ABB RobotStudio station: Project2.rsstnx

Station Project2 (saved by RobotStudio 24.3.10885.0)
Controller Controller1
  mechanical unit ROB_1: IRB2600_12_185__02, 6 joints, base frame (0, 0, 0) mm
Layout (positions relative to the parent item):
  - Ratata [mechanism] at (1018.61, 0, 1417.5) mm, rotated rx 180 ry 60 rz 180 deg
      TCP Ratata at (0, -50, 190) mm, rotated rx 30 ry 0 rz 0 deg
      links: Group_2
  - IRB2600_12_185__02 [mechanism, from %ABB.RobotStudio.Models.IRB2600%\IRB2600_12_185_G_02.rslib] at (0, 0, 0) mm; joint values [0, 0, 0, 0, 0.5236, 0] (rad or m)
  - Part_6 [part], size 214.9 x 213.7 x 0 mm
  - Part_7 [part] at (135.15, 0, 0) mm, size 214.9 x 213.7 x 400 mm
  - Part_14 [part], size 168 x 171.3 x 400 mm
  - Part_16 [part] at (400, 920.93, 1412.57) mm, rotated rx 0 ry 90 rz 0 deg, size 214.9 x 213.7 x 400 mm
  - Part_17 [part], size 1500 x 10 x 1500 mm
Attachment: Ratata is attached to IRB2600_12_185__02 / Link6
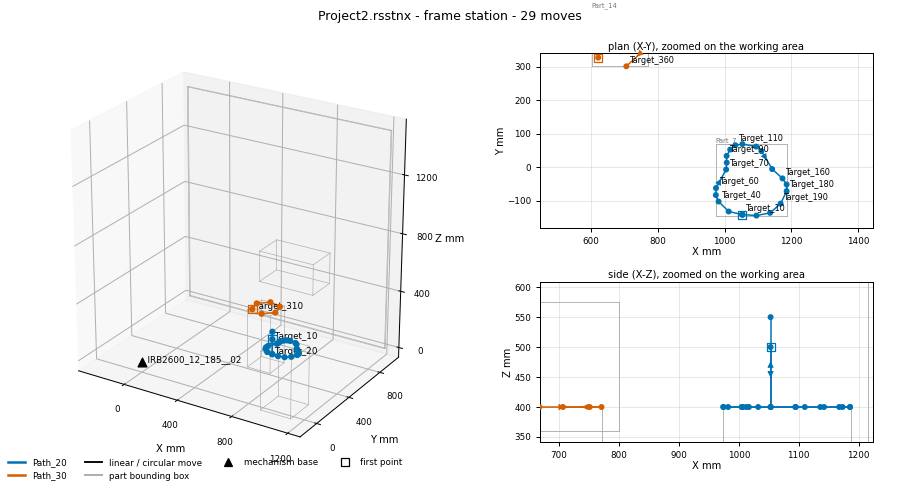
[picture p0: tool path of Project2.rsstnx in frame station, 29 of 29 moves have a stored position in this frame; points joined in program order, loops and branches not executed]
Targets, tools, work objects and paths stored in the station, written as RAPID:
! task T_ROB1
MODULE CalibData
  PERS tooldata Ratata:=[TRUE,[[0,-50,190],[0.965925826,0.258819045,0,0]],[1,[0,0,90],[1,0,0,0],0,0,0]];
  TASK PERS wobjdata Workobject_1:=[FALSE,TRUE,"",[[622.473,327.081,400],[1,0,0,0]],[[0,0,0],[1,0,0,0]]];
ENDMODULE

! task T_ROB1
MODULE Module1
  CONST jointtarget JointTarget_1:=[[0,0,0,0,0,0],[9E+09,9E+09,9E+09,9E+09,9E+09,9E+09]];
  CONST robtarget Target_10:=[[1053.028483888,-141.83,500],[0,0.048639314,0.998816408,0],[0,0,0,0],[9E+09,9E+09,9E+09,9E+09,9E+09,9E+09]];
  CONST robtarget Target_20:=[[1053.028483888,-141.83,400],[0,0.048639314,0.998816408,0],[-1,0,-1,0],[9E+09,9E+09,9E+09,9E+09,9E+09,9E+09]];
  CONST robtarget Target_30:=[[1012.393593189,-132.667043204,400],[0,0.247498073,0.968888386,0],[-1,0,-1,0],[9E+09,9E+09,9E+09,9E+09,9E+09,9E+09]];
  CONST robtarget Target_40:=[[982.192356429,-102.911473019,400],[0,0.483619111,0.875278559,0],[-1,0,-1,0],[9E+09,9E+09,9E+09,9E+09,9E+09,9E+09]];
  CONST robtarget Target_50:=[[973.974019148,-83.529915198,400],[0,0.630396667,0.776273175,0],[-1,1,-1,0],[9E+09,9E+09,9E+09,9E+09,9E+09,9E+09]];
  CONST robtarget Target_60:=[[974.486081612,-62.744242155,400],[0,0.783865496,0.620930659,0],[-1,2,-2,0],[9E+09,9E+09,9E+09,9E+09,9E+09,9E+09]];
  CONST robtarget Target_70:=[[1004.654113735,-7.369996452,400],[0,0.83364436,0.552301621,0],[0,3,-2,0],[9E+09,9E+09,9E+09,9E+09,9E+09,9E+09]];
  CONST robtarget Target_80:=[[1006.554953292,13.24883335,400],[0,0.617780056,0.786350941,0],[-1,1,-1,0],[9E+09,9E+09,9E+09,9E+09,9E+09,9E+09]];
  CONST robtarget Target_90:=[[1006.144920769,33.417655307,400],[0,0.829177231,0.558985796,0],[0,3,-2,0],[9E+09,9E+09,9E+09,9E+09,9E+09,9E+09]];
  CONST robtarget Target_100:=[[1016.902942171,52.408008378,400],[0,0.878010395,0.478641563,0],[0,3,-2,0],[9E+09,9E+09,9E+09,9E+09,9E+09,9E+09]];
  CONST robtarget Target_110:=[[1032.336239923,65.35895098,400],[0,0.986205127,0.165527784,0],[0,3,-2,0],[9E+09,9E+09,9E+09,9E+09,9E+09,9E+09]];
  CONST robtarget Target_120:=[[1053.446161766,68.778243604,400],[0,0.99965304,0.026340074,0],[0,3,-2,0],[9E+09,9E+09,9E+09,9E+09,9E+09,9E+09]];
  CONST robtarget Target_130:=[[1094.310928385,61.39343752,400],[0,0.971088832,-0.238718412,0],[0,3,-2,0],[9E+09,9E+09,9E+09,9E+09,9E+09,9E+09]];
  CONST robtarget Target_140:=[[1110.161148991,47.833471517,400],[0,0.897820327,-0.440361966,0],[0,3,-2,0],[9E+09,9E+09,9E+09,9E+09,9E+09,9E+09]];
  CONST robtarget Target_150:=[[1142.282150365,-5.867956748,400],[0,0.940674196,-0.33931115,0],[0,3,-2,0],[9E+09,9E+09,9E+09,9E+09,9E+09,9E+09]];
  CONST robtarget Target_160:=[[1173.132567714,-33.754311671,400],[0,0.896740471,-0.442556808,0],[0,3,-2,0],[9E+09,9E+09,9E+09,9E+09,9E+09,9E+09]];
  CONST robtarget Target_170:=[[1185.623777539,-51.793265608,400],[0,0.845978482,-0.533217036,0],[-1,3,-2,0],[9E+09,9E+09,9E+09,9E+09,9E+09,9E+09]];
  CONST robtarget Target_180:=[[1185.639297263,-71.745848185,400],[0,-0.586154613,0.810199216,0],[-1,4,-1,0],[9E+09,9E+09,9E+09,9E+09,9E+09,9E+09]];
  CONST robtarget Target_190:=[[1167.562709351,-109.141891193,400],[0,-0.422507005,0.906359658,0],[-1,4,-1,0],[9E+09,9E+09,9E+09,9E+09,9E+09,9E+09]];
  CONST robtarget Target_200:=[[1136.030927079,-136.731454767,400],[0,-0.222736348,0.97487872,0],[-1,4,-1,0],[9E+09,9E+09,9E+09,9E+09,9E+09,9E+09]];
  CONST robtarget Target_210:=[[1095.203821678,-144.904989424,400],[0,-0.003413263,0.999994175,0],[-1,4,-1,0],[9E+09,9E+09,9E+09,9E+09,9E+09,9E+09]];
  CONST robtarget Target_220:=[[1053.028483888,-141.83,400],[0,0.048639314,0.998816408,0],[0,0,0,0],[9E+09,9E+09,9E+09,9E+09,9E+09,9E+09]];
  CONST robtarget Target_230:=[[1053.028483888,-141.83,550],[0,0.048639314,0.998816408,0],[0,0,0,0],[9E+09,9E+09,9E+09,9E+09,9E+09,9E+09]];
  CONST robtarget Target_290:=[[-19.683,85.658,0],[0,1,0,0],[0,0,0,0],[9E+09,9E+09,9E+09,9E+09,9E+09,9E+09]];
  CONST robtarget Target_300:=[[560.683986041,-377.081,922.5],[0.482962913,0.129409523,0.836516304,-0.224143868],[0,-1,0,0],[9E+09,9E+09,9E+09,9E+09,9E+09,9E+09]];
  CONST robtarget Target_310:=[[0,0,0],[0,0.622915127,0.782289425,0],[0,0,0,0],[9E+09,9E+09,9E+09,9E+09,9E+09,9E+09]];
  CONST robtarget Target_320:=[[-19.683271052,85.657574479,0],[0,0.622915127,0.782289425,0],[0,0,0,0],[9E+09,9E+09,9E+09,9E+09,9E+09,9E+09]];
  CONST robtarget Target_330:=[[44.656728948,145.532574479,0],[0,0.930605037,0.366024952,0],[0,0,0,0],[9E+09,9E+09,9E+09,9E+09,9E+09,9E+09]];
  CONST robtarget Target_340:=[[128.68,119.75,0],[0,0.988940079,-0.148315612,0],[0,0,0,0],[9E+09,9E+09,9E+09,9E+09,9E+09,9E+09]];
  CONST robtarget Target_350:=[[148.363271052,34.092425521,0],[0,0.782289425,-0.622915127,0],[0,0,0,0],[9E+09,9E+09,9E+09,9E+09,9E+09,9E+09]];
  CONST robtarget Target_360:=[[84.023271052,-25.782574479,0],[0,-0.366024952,0.930605037,0],[0,0,0,0],[9E+09,9E+09,9E+09,9E+09,9E+09,9E+09]];
  PROC Path_10()
  ENDPROC
  PROC Path_20()
    MoveL Target_10,v1000,z100,Ratata\WObj:=wobj0;
    MoveL Target_20,v1000,z100,Ratata\WObj:=wobj0;
    MoveL Target_30,v1000,z100,Ratata\WObj:=wobj0;
    MoveL Target_40,v1000,z100,Ratata\WObj:=wobj0;
    MoveL Target_50,v1000,z100,Ratata\WObj:=wobj0;
    MoveL Target_60,v1000,z100,Ratata\WObj:=wobj0;
    MoveL Target_70,v1000,z100,Ratata\WObj:=wobj0;
    MoveL Target_80,v1000,z100,Ratata\WObj:=wobj0;
    MoveL Target_90,v1000,z100,Ratata\WObj:=wobj0;
    MoveL Target_100,v1000,z100,Ratata\WObj:=wobj0;
    MoveL Target_110,v1000,z100,Ratata\WObj:=wobj0;
    MoveL Target_120,v1000,z100,Ratata\WObj:=wobj0;
    MoveL Target_130,v1000,z100,Ratata\WObj:=wobj0;
    MoveL Target_140,v1000,z100,Ratata\WObj:=wobj0;
    MoveL Target_150,v1000,z100,Ratata\WObj:=wobj0;
    MoveL Target_160,v1000,z100,Ratata\WObj:=wobj0;
    MoveL Target_170,v1000,z100,Ratata\WObj:=wobj0;
    MoveL Target_180,v1000,z100,Ratata\WObj:=wobj0;
    MoveL Target_190,v1000,z100,Ratata\WObj:=wobj0;
    MoveL Target_200,v1000,z100,Ratata\WObj:=wobj0;
    MoveL Target_210,v1000,z100,Ratata\WObj:=wobj0;
    MoveL Target_220,v1000,z100,Ratata\WObj:=wobj0;
    MoveL Target_230,v1000,z100,Ratata\WObj:=wobj0;
  ENDPROC
  PROC Path_30()
    MoveL Target_310,v1000,z100,Ratata\WObj:=Workobject_1;
    MoveL Target_320,v1000,z100,Ratata\WObj:=Workobject_1;
    MoveL Target_330,v1000,z100,Ratata\WObj:=Workobject_1;
    MoveL Target_340,v1000,z100,Ratata\WObj:=Workobject_1;
    MoveL Target_350,v1000,z100,Ratata\WObj:=Workobject_1;
    MoveL Target_360,v1000,z100,Ratata\WObj:=Workobject_1;
  ENDPROC
ENDMODULE

